(* CODESYS project MID_COM_Demo.project

Project tree, tasks and I/O mapping:
  Device : Changsha Xiangji-ARM Cortex A9(xilinx zynq7000)-linux, Changsha Xiangji Hiden Technology Co.Ltd, version 3.5.10.20
    application Application
      libraries: Standard, * (System); VisuDialogs, * (System); CAA SerialCom, * (CAA Technical Workgroup); CAA Types Extern, * (CAA Technical Workgroup)
      task MainTask (cyclic, interval 4 ms, priority 1) calls COM_SERIAL
      task VISU_TASK (cyclic, interval 100 ms, priority 31) calls VisuElems.Visu_Prg
      RS485/
        program COM_SERIAL [ST]
      global variables GVL
      visualisation COM_test_Visua
      text list COM_Type_TextList
    SoftMotion General Axis Pool
  text list GlobalTextList
*)

// Device/Application/GVL
{attribute 'qualified_only'}
{attribute 'qualified_only'}


VAR_GLOBAL

	
	Writebuffer:			ARRAY[1..14] OF BYTE;
	Readbuffer: 			ARRAY[1..16] OF BYTE;
	COMWritebuffer:			ARRAY[1..14] OF STRING;
	COMReadbuffer: 			ARRAY[1..16] OF STRING;
	send_serial :BYTE := 0;
	pwm_1A:BOOL := FALSE;

	cmdSend:BOOL := FALSE;
	recvOk:BOOL := FALSE;

	ComType:INT:=0;



END_VAR

// Device/Application/RS485/COM_SERIAL
PROGRAM COM_SERIAL
VAR		
	Com1Params: 			ARRAY [1..7] OF COM.PARAMETER;	(* Settings to communicate with the COM Port *)
	hCom: 					CAA.HANDLE;
	ComOpen: 				COM.Open;
	ComClose: 				COM.Close;
	ComWrite: 				COM.Write;
	ComRead: 				COM.Read;	
	
	//Writebuffer: 			STRING:= 'Hello! zhouqin';

	Snd_Cnt:				CAA.SIZE;

	Rcv_Cnt: 				CAA.SIZE;
	xCom1CloseError: 		BOOL;
	xCom1WriteError: 		BOOL;
	xCom1ReadError: 		BOOL;
	xError:					BOOL;
	
	uiComState: INT := 0;
	uiComState_MC20: INT := 0;
	ComID:USINT:=4;//串口号为3
	ComID_MC20:USINT:=3;//串口号为4

	cmdSend:BOOL := FALSE;
	COMWritebufsum: 	    STRING(200):='ABCDE';
	COMReadbufsum: 			STRING(1000):='';
	COMReadbufsum1: 			STRING(1000);
	COMWritebufsum_MC20: 	    STRING(200):='';
	COMReadbufsum_MC20: 			STRING(200);
//	boot_flag: INT;
	ton2:TON;
	size:CAA.SIZE;
	
    at_GPSOPEN_cmd :STRING := 'AT+QGNSSC=1';
	at_ask_buffer1 :STRING(1000);
	at_ask_buffer2 :STRING(1000);
	at_ask_buffer3 :STRING(1000);
	at_ask_buffer4 :STRING(1000);
	at_ask_buffer5:STRING(1000);
	at_ask_buffer6 :STRING(1000);
	at_GPSREAD_cmd :STRING := 'AT+QGNSSRD="NMEA/RMC"';
	at_GPSREAD_buffer :STRING;
	ComType:INT:=0;
	ComReadSize:INT;
	
END_VAR



CASE uiComState OF
	0:
	Com1Params[1].udiParameterId := COM.CAA_Parameter_Constants.udiPort;
	Com1Params[1].udiValue := ComID; 
	Com1Params[2].udiParameterId := COM.CAA_Parameter_Constants.udiBaudrate;
	Com1Params[2].udiValue := 115200;
	Com1Params[3].udiParameterId := COM.CAA_Parameter_Constants.udiParity;
	Com1Params[3].udiValue := INT_TO_UINT(COM.PARITY.NONE);
	Com1Params[4].udiParameterId := COM.CAA_Parameter_Constants.udiStopBits;
	Com1Params[4].udiValue := INT_TO_UINT(COM.STOPBIT.ONESTOPBIT);
	Com1Params[5].udiParameterId := COM.CAA_Parameter_Constants.udiTimeout;
	Com1Params[5].udiValue := 0;
	Com1Params[6].udiParameterId := COM.CAA_Parameter_Constants.udiByteSize;
	Com1Params[6].udiValue := 8;
	Com1Params[7].udiParameterId := COM.CAA_Parameter_Constants.udiBinary;
	Com1Params[7].udiValue := 0;					
	ComOpen(xExecute := TRUE, usiListLength:=UINT_TO_USINT(SIZEOF(Com1Params)/SIZEOF(COM.PARAMETER)),pParameterList:= ADR(Com1Params),hCom=> hCom);			
	IF ComOpen.xError THEN
		uiComState := 32767;
	ELSIF ComOpen.xDone THEN
		uiComState := 1;
		ComWrite(xExecute := FALSE,hCom:= hCom);	
		ComRead(xExecute := FALSE,hCom:= hCom);
	END_IF
	
	1:

	IF cmdSend  THEN
		ComWrite(xExecute := TRUE,hCom:= hCom,pBuffer:= ADR(COMWritebufsum),szSize:= ANY_TO_UINT(len(COMWritebufsum)));		
		IF ComWrite.xError THEN
			uiComState := 32767;
		END_IF
		IF ComWrite.xDone THEN		
			ComWrite(xExecute := FALSE);
			uiComState := 2;
			gvl.send_serial := gvl.send_serial + 1;
			gvl.cmdSend := FALSE;
			gvl.recvOk := FALSE;
		END_IF
	END_IF
	
	
	
   2:
	TON2(IN:=TRUE,PT:=T#200MS);
		IF TON2.Q=TRUE THEN
                uiComState := 3;
				TON2(IN:=FALSE,PT:=T#200MS);
		END_IF
	
	3:
	
    ComRead(xExecute := FALSE,hCom:= hCom, pBuffer:= ADR(COMReadbufsum), szBuffer:= SIZEOF(COMReadbufsum));	
	ComRead.xExecute := TRUE;//给xExecute制造一个上升沿，读串口命令才能被调用一次
	
    IF ComRead.xError THEN
		uiComState := 32767;
	END_IF
	
	255:
	
	32767:	
END_CASE



ComRead(xExecute := TRUE,hCom:= hCom, pBuffer:= ADR(COMReadbufsum), szBuffer:= SIZEOF(COMReadbufsum));	
ComReadSize:=ANY_TO_INT(ComRead.szSize);
IF ComReadSize<>0 THEN
	COMReadbufsum1:=left(COMReadbufsum,ComReadSize);
ELSE
	COMReadbufsum:=COMReadbufsum1;
END_IF

END_PROGRAM

// Device/Application/COM_test_Visua
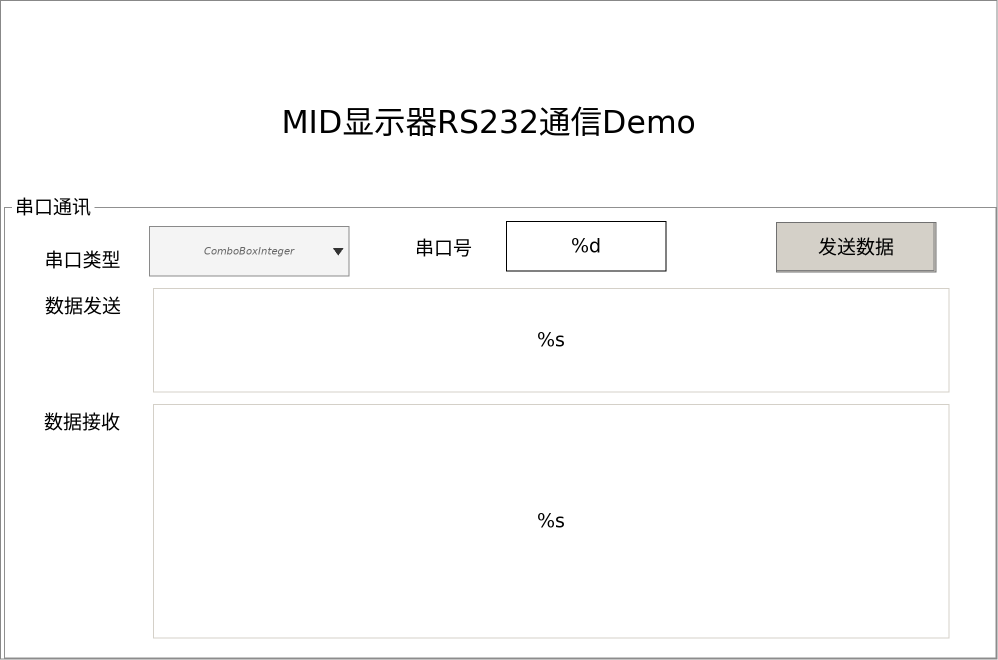
VISUALIZATION COM_test_Visua  // 998x660
    GroupBox (4,199 992x459), "串口通讯"
        Label (5,30 147x62), "串口类型"
        Label (4,76 150x62), "数据发送"
        Button (772,23 160x50), "发送数据"
            OnMouseDown: execute { COM_SERIAL.uiComState:=0; COM_SERIAL.cmdSend:=true; }
        Label (17,191 122x64), "数据接收"
        ComboBoxInteger (145,27 200x50), variable: GVL.ComType, text list: 'COM_Type_TextList'
        Label (366,18 147x62), "串口号"
        Rectangle (502,22 160x50), "%d", text variable: COM_SERIAL.ComID
            OnMouseDown: write the text variable via VisuDialogs.Numpad, min 0, max 255
        Textfield (149,89 796x104), "%s", text variable: COM_SERIAL.COMWritebufsum
            OnMouseClick: write COM_SERIAL.COMWritebufsum via Default
    Textfield (153,404 796x234), "%s", text variable: COM_SERIAL.COMReadbufsum1
    Label (202,79 574x86), "MID显示器RS232通信Demo"
END_VISUALIZATION

(* text list COM_Type_TextList (id | default)
  0 | RS232
  1 | RS485
   |  *)
